// TIA Portal V18 export
DATA_BLOCK "Simulation_Data_1_DB"   // DB3
VERSION : 0.1
// stored: AutoNumber true, DBAccessibleFromOPCUA true, DBAccessibleFromWebserver true, InstanceOfName Simulation_Data_1, InstanceOfType FB
"Simulation_Data_1"
   // VAR
   //    Old_Clock : Bool;
   //    i : Int;
   // END_VAR
BEGIN
END_DATA_BLOCK
